// TIA Portal V20 export
DATA_BLOCK "BK31"   // DB279
// stored: MemoryReserve 100
   VAR
      "X10-1.ANODE MAIN P&P1-1 VACUUM ON" : Bool := FALSE;
      "X10-2.ANODE MAIN P&P1-1 VACUUM OFF" : Bool := FALSE;
      "X12-1.ANODE MAIN P&P2-1 VACUUM ON" : Bool := FALSE;
      "X12-2.ANODE MAIN P&P2-1 VACUUM OFF" : Bool := FALSE;
      "X14-1.ANODE MAIN NG P&P VACUUM ON" : Bool := FALSE;
      "X14-2.ANODE MAIN NG P&P VACUUM OFF" : Bool := FALSE;
      "X16-1.ANODE ALIGN TABLE VACUUM ON" : Bool := FALSE;
      "X16-2.ANODE ALIGN TABLE VACUUM OFF" : Bool := FALSE;
   END_VAR
BEGIN
END_DATA_BLOCK
